// This function has been automatically generated from the project information.
{attribute 'signature_flag' := '1073741824'}
{attribute 'TcGenerated'}
{attribute 'no-analysis'}
FUNCTION F_GetTitle : WSTRING
VAR_INPUT
	
END_VAR

F_GetTitle := "FsTime";

END_FUNCTION

(* stored: Version 1.1.0.1
   POU F_GetTitle: Id {deb0ef93-b05d-4431-8317-dd545e78e1f0}, SpecialFunc None *)
